Fanuc KAREL source: NC0062.KL

-- PROVISIONAL review KL for V940-1; original PC SHA256 173547eddf9d1fd233e4fab82c58c80090f50167a361e60e51c08ff2da83eac1
-- Incomplete behavior may be omitted. Consult companion uncertainty JSON. Do not deploy.
PROGRAM NC0062
%NOLOCKGROUP
-- UNRESOLVED_LOCAL_POOL 2 cells at code offset 3; source declarations unknown
-- DIRECT_LOCAL_WORD_ACCESS alone does not prove INTEGER, REAL, or BOOLEAN
BEGIN
  -- V9_EXPOSED_INDEXED_TABLE_HINT layout=0001; 2 counted words exposed once; source arms/runtime held
  -- V9_FOOTER_20_HINT 1 numerical footer links; VM transfer unproved
  -- UNRESOLVED_PC offsets 0-8; opcodes 2B,2C,7B
  -- UNRESOLVED_PC offsets 13-20; opcodes 9D,23
  -- UNRESOLVED_PC offsets 25-54; opcodes 9D,23,9E,2E,22,7A
  -- UNRESOLVED_PC offsets 59-73; opcodes 21,9D,52,23
  -- UNRESOLVED_PC offsets 78-93; opcodes 20,2C,23
  -- UNRESOLVED_PC offsets 98-102; opcodes 7F
  -- UNRESOLVED_PC offsets 107-111; opcodes 27,AA
  -- UNRESOLVED_PC offsets 116-120; opcodes 7F
END NC0062
